Staubli VAL3: Day4.pjx

--- Day4.pjx ---
Parameters version=s8.13.1Cs9_BS2800 stackSize=5000 millimeterUnit=true
Program file=calc_WinningNumber.pgx
Program file=check_table.pgx
Program file=findNumberInMatrix.pgx
Program file=init_tables.pgx
Program file=size_tables.pgx
Program file=start.pgx
Program file=stop.pgx
Data file=Day4.dtx
Library alias=util path=Disk://helpers/helpers.pjx
Library alias=math path=Disk://math/math.pjx
Library alias=str path=Disk://string/string.pjx
Type name=lists path=Disk://types/lists/lists.pjx
Type name=lists_num path=Disk://types/lists_num/lists_num.pjx
Type name=table path=./table/table.pjx

--- Day4.dtx ---
string sInput
lists lResult
  [0]
    string sString
num nResult
table tTable
  [0]
    num nMatrix[1 1]
lists lLine
  [0]
    string sString
num nBingoNumbers1
num nBingoNumbers2
num nBingoNumbers
table tTable_remove
  [0]
    num nMatrix[1 1]
table tTable_empty
  [0]
    num nMatrix[1 1]
num nResultRow
num nResultCol
bool bWinner
num nIndexX
num nIndexY
bool bFound
bool bHasWon

--- start.pgx ---
program start()
  local num l_nTable
  local num l_nBingoIndex
  local num l_nElement
  local num l_nResult
  local bool l_bAllWon
begin

  // read file
  call util:readFile("Disk://input_day4.txt", sInput)
  // sInput[0] = "26,38,2,15,....."

  // parse Bingo-Numbers
  call str:splitString(sInput[0],"," ,lResult)
  call util:vec2num(lResult.sString[0], nBingoNumbers1)

  call str:splitString(sInput[1],"," ,lResult)
  call util:vec2num(lResult.sString[0], nBingoNumbers2)

  call util:mergeVectors(nBingoNumbers1,nBingoNumbers2, nBingoNumbers)

  // Now nBingoNumbers

  // parse tables
  delete(lResult[1])
  delete(lResult[0])

  // prepare tables
  call size_tables()
  call init_tables()

  // TEST
  //call check_table(tTable_empty.nMatrix, bWinner)

  // PUZZLE 1
  l_nBingoIndex = 0
  bWinner = false
  while bWinner == false
    for l_nTable = 0 to size(tTable)-1

      // check if current bingo number is in matrix
      call findNumberInMatrix(tTable[l_nTable].nMatrix, nBingoNumbers[l_nBingoIndex], nIndexX, nIndexY, bFound)

      // if yes: remove it in tTable_remove and add 1 to tTable_empty on same position
      if bFound
        for l_nElement = 0 to size(nIndexX)-1
          tTable_remove[l_nTable].nMatrix[nIndexX[l_nElement], nIndexY[l_nElement]] = 0
          tTable_empty[l_nTable].nMatrix[nIndexX[l_nElement], nIndexY[l_nElement]] = 1
        endFor
      endIf

      // check if we have a winner!
      call check_table(tTable_empty[l_nTable].nMatrix, bWinner)

      if bWinner
        call calc_WinningNumber(tTable_remove[l_nTable].nMatrix, nBingoNumbers[l_nBingoIndex], l_nResult)
        call util:printNum(l_nResult)
        // to break the for loop
        l_nTable = size(tTable)+1
      endIf

    endFor

    l_nBingoIndex = l_nBingoIndex +1
  endWhile

  // 58374

  // PUZZLE 2

  call size_tables()
  call init_tables()

  resize(bHasWon,1,1)
  bHasWon=false
  resize(bHasWon,1,size(tTable))

  l_nBingoIndex = 0
  bWinner = false
  while bWinner == false
    for l_nTable = 0 to size(tTable)-1

      // check if current bingo number is in matrix
      call findNumberInMatrix(tTable[l_nTable].nMatrix, nBingoNumbers[l_nBingoIndex], nIndexX, nIndexY, bFound)

      // if yes: remove it in tTable_remove and add 1 to tTable_empty on same position
      if bFound
        for l_nElement = 0 to size(nIndexX)-1
          tTable_remove[l_nTable].nMatrix[nIndexX[l_nElement], nIndexY[l_nElement]] = 0
          tTable_empty[l_nTable].nMatrix[nIndexX[l_nElement], nIndexY[l_nElement]] = 1
        endFor
      endIf

      // check if we have a winner!
      call check_table(tTable_empty[l_nTable].nMatrix, bWinner)

      if bWinner and bHasWon[l_nTable] ==false

        bHasWon[l_nTable] = true

        call util:allBool(bHasWon, l_bAllWon)
        if l_bAllWon
          call calc_WinningNumber(tTable_remove[l_nTable].nMatrix, nBingoNumbers[l_nBingoIndex], l_nResult)
          call util:printNum(l_nResult)
          // to break the for loop
          l_nTable = size(tTable)+1
        endIf

      endIf

    endFor
    if bWinner and !l_bAllWon
      bWinner = false
    endIf

    l_nBingoIndex = l_nBingoIndex +1
  endWhile

  // 11377


end

--- calc_WinningNumber.pgx ---
program calc_WinningNumber(num& x_nCurrentMatrix[] (dimensions=2), num x_nCurrentNumber, num& x_nRESULT)
  local num l_nX
  local num l_nY
begin

  //resize(x_nRESULT,1,1)
  x_nRESULT = 0
  for l_nX = 0 to size(x_nCurrentMatrix,1)-1
    for l_nY = 0 to size(x_nCurrentMatrix,2)-1
      x_nRESULT = x_nRESULT + x_nCurrentMatrix[l_nX, l_nY]
    endFor
  endFor

  x_nRESULT = x_nRESULT*x_nCurrentNumber

end

--- check_table.pgx ---
program check_table(num& x_nInput[] (dimensions=2), bool& x_bResult)
  local num l_nElement
begin

  call util:rowSum(x_nInput, nResultRow)
  call util:colSum(x_nInput, nResultCol)
  x_bResult = false
  //check if ANY row or col is 0!

  for l_nElement = 0 to size(nResultRow)-1
    if nResultRow[l_nElement] == size(nResultRow)
      x_bResult = true
      return
    endIf
  endFor

  for l_nElement = 0 to size(nResultCol)-1
    if nResultCol[l_nElement] == size(nResultCol)
      x_bResult = true
      return
    endIf
  endFor


end

--- findNumberInMatrix.pgx ---
program findNumberInMatrix(num& x_nInput[] (dimensions=2), num x_nNumber, num& x_nIndexX[], num& x_nIndexY[], bool& x_bFound)
  local num l_nX
  local num l_nY
  local num l_nFoundCounter
begin

  resize(x_nIndexX,1,1)
  x_nIndexX = -1
  resize(x_nIndexY,1,1)
  x_nIndexY = -1
  x_bFound = false

  for l_nX = 0 to size(x_nInput,1)-1
    for l_nY = 0 to size(x_nInput,2)-1

      if x_nNumber == x_nInput[l_nX,l_nY]
        x_bFound = true
        if l_nFoundCounter != 0
          append(x_nIndexX)
          append(x_nIndexY)
        endIf

        x_nIndexX[l_nFoundCounter] = l_nX
        x_nIndexY[l_nFoundCounter] = l_nY
        l_nFoundCounter = l_nFoundCounter + 1
      endIf

    endFor
  endFor


end

--- init_tables.pgx ---
program init_tables()
  local num l_nElement
  local num l_nMatrixEntry
  local num l_nRow
  local num l_nTable
  local string l_sLine
begin

  l_nTable = 0
  for l_nElement = 1 to size(lResult)

    if l_nElement %6 != 0
      l_sLine = lResult[l_nElement-1].sString
      call str:splitString(l_sLine," " ,lLine)
      call util:vec2num(lLine.sString,nResult)
      for l_nMatrixEntry = 0 to 4
        tTable[l_nTable].nMatrix[l_nRow, l_nMatrixEntry] = nResult[l_nMatrixEntry]
        tTable_remove[l_nTable].nMatrix[l_nRow, l_nMatrixEntry] = nResult[l_nMatrixEntry]
      endFor
      l_nRow = l_nRow+1
    else
      l_nRow = 0
      l_nTable = l_nTable + 1
      append(tTable)
      resize(tTable[l_nTable].nMatrix,1,5)
      resize(tTable[l_nTable].nMatrix,2,5)
      append(tTable_remove)
      resize(tTable_remove[l_nTable].nMatrix,1,5)
      resize(tTable_remove[l_nTable].nMatrix,2,5)
      append(tTable_empty)
      resize(tTable_empty[l_nTable].nMatrix,1,5)
      resize(tTable_empty[l_nTable].nMatrix,2,5)
    endIf
  endFor

end

--- size_tables.pgx ---
program size_tables()
begin

  // input tables
  resize(tTable.nMatrix,1,1)
  resize(tTable.nMatrix,2,1)
  resize(tTable,1,1)
  tTable.nMatrix[0,0] = 0
  resize(tTable.nMatrix,1,5)
  resize(tTable.nMatrix,2,5)

  // table to remove numbers with 0s
  resize(tTable_remove.nMatrix,1,1)
  resize(tTable_remove.nMatrix,2,1)
  resize(tTable_remove,1,1)
  tTable_remove.nMatrix[0,0] = 0
  resize(tTable_remove.nMatrix,1,5)
  resize(tTable_remove.nMatrix,2,5)

  // table_empty to fill with 1s
  resize(tTable_empty.nMatrix,1,1)
  resize(tTable_empty.nMatrix,2,1)
  resize(tTable_empty,1,1)
  tTable_empty.nMatrix[0,0] = 0
  resize(tTable_empty.nMatrix,1,5)
  resize(tTable_empty.nMatrix,2,5)


end
